(* CODESYS project CtaAppKelvinminuten_1.0.0.0.library
   Description: Kelvinminuten Library der CTA
   Version: 1.0.0.0
   Title: CtaAppKelvinminuten
   Author: SIS
   Company: CTA
   Placeholder: CtaAppKelvinminuten
   DocFormat: reStructuredText
   CompiledLibraryCompatibilityVersion: CODESYS V3.5 SP16 Patch 3
   LanguageModelAttribute: qualified-access-only
   DefaultNamespace: CtaAppKelvinminuten

Project tree, tasks and I/O mapping:
  libraries: CmpBitmapPool, 3.5.17.0 (System); CtaVisSymbols, 1.0.0.0 (CTA); CtaSysConfig, 1.0.0.0 (CTA); CtaAppTime, 1.0.0.0 (CTA); VisuSymbols, 4.5.0.0 (System)
  40 Visualizations/
    visualisation visKelvinminuten
    visualisation popUpKelvinminuten
  30 Program Organization Units/
    function block fbKelvinminuten [ST]: actParameter
  00000000-0000-0000-0000-000000000000|D:\CoDeSys\LibrariesV3\trunk\Intern\CAA\CAA Template\3.4.0.0 draft\Placeholder.xml
  00000000-0000-0000-0000-000000000000|D:\CoDeSys\LibrariesV3\trunk\Intern\CAA\CAA Template\3.2.0.3 draft\Prefix.pdf
  00000000-0000-0000-0000-000000000000|D:\CoDeSys\LibrariesV3\trunk\Intern\CAA\CAA Template\3.5.2.0 draft\Placeholder.xml
  20 Structs/
    data type scParameter
    data type enState
  50 Images/
  10 Documenation/
    global variables VersionHistory
    global variables readMe
  21 Interface/
  11 Library Parameter/
  12 Konstanten/
  60 Textlisten/
  13 Globale Variablen/
  5ce3da45-db07-42e7-a21c-a00fff4ed8f6|Icons\alert.svg
  5ce3da45-db07-42e7-a21c-a00fff4ed8f6|Icons\arrow-down.svg
  5ce3da45-db07-42e7-a21c-a00fff4ed8f6|Icons\arrow-down_square.svg
  5ce3da45-db07-42e7-a21c-a00fff4ed8f6|Icons\arrow-left_solo_black.svg
  5ce3da45-db07-42e7-a21c-a00fff4ed8f6|Icons\arrow-right_solo_black.svg
  5ce3da45-db07-42e7-a21c-a00fff4ed8f6|Icons\arrow-up.svg
  5ce3da45-db07-42e7-a21c-a00fff4ed8f6|Icons\calendar-range.svg
  5ce3da45-db07-42e7-a21c-a00fff4ed8f6|Icons\check.svg
  5ce3da45-db07-42e7-a21c-a00fff4ed8f6|Icons\clock-outline.svg
  5ce3da45-db07-42e7-a21c-a00fff4ed8f6|Icons\close_solo_black.svg
  5ce3da45-db07-42e7-a21c-a00fff4ed8f6|Icons\CtaInfo.svg
  5ce3da45-db07-42e7-a21c-a00fff4ed8f6|Icons\database_black.svg
  5ce3da45-db07-42e7-a21c-a00fff4ed8f6|Icons\delete_solo_black.svg
  5ce3da45-db07-42e7-a21c-a00fff4ed8f6|Icons\engine.svg
  5ce3da45-db07-42e7-a21c-a00fff4ed8f6|Icons\front_hand_Black.svg
  5ce3da45-db07-42e7-a21c-a00fff4ed8f6|Icons\front_hand_Yellow_Off.svg
  5ce3da45-db07-42e7-a21c-a00fff4ed8f6|Icons\gear.svg
  5ce3da45-db07-42e7-a21c-a00fff4ed8f6|Icons\home.svg
  5ce3da45-db07-42e7-a21c-a00fff4ed8f6|Icons\information-variant.svg
  5ce3da45-db07-42e7-a21c-a00fff4ed8f6|Icons\lightning-bolt-circle.svg
  5ce3da45-db07-42e7-a21c-a00fff4ed8f6|Icons\message.svg
  5ce3da45-db07-42e7-a21c-a00fff4ed8f6|Icons\message-alert-variant.svg
  5ce3da45-db07-42e7-a21c-a00fff4ed8f6|Icons\minus_solo_black.svg
  5ce3da45-db07-42e7-a21c-a00fff4ed8f6|Icons\plus_solo_black.svg
  5ce3da45-db07-42e7-a21c-a00fff4ed8f6|Icons\power_solo_black.svg
  5ce3da45-db07-42e7-a21c-a00fff4ed8f6|Icons\refresh_solo_black.svg
  5ce3da45-db07-42e7-a21c-a00fff4ed8f6|Icons\SearchFilter.svg
  5ce3da45-db07-42e7-a21c-a00fff4ed8f6|Icons\signal-celular-alt.svg
  5ce3da45-db07-42e7-a21c-a00fff4ed8f6|Icons\toggle-switch.svg
  5ce3da45-db07-42e7-a21c-a00fff4ed8f6|Icons\Modbus_Organization_Logo.svg
  5ce3da45-db07-42e7-a21c-a00fff4ed8f6|Icons\CheckboxUnchecked_withe.svg
  5ce3da45-db07-42e7-a21c-a00fff4ed8f6|Icons\lock_open_black.svg
  5ce3da45-db07-42e7-a21c-a00fff4ed8f6|Icons\check_green.svg
  5ce3da45-db07-42e7-a21c-a00fff4ed8f6|Icons\filter_black.svg
  5ce3da45-db07-42e7-a21c-a00fff4ed8f6|Icons\CtaLogo.png
  5ce3da45-db07-42e7-a21c-a00fff4ed8f6|Icons\Grafana_Logo.svg
  5ce3da45-db07-42e7-a21c-a00fff4ed8f6|Icons\hourglass_top.svg
  text list GlobalTextList
*)

// 20 Structs/scParameter
TYPE scParameter :
	STRUCT
		fbrKmZuschalt   : CtaSysConfig.fbREAL;
		fbrKmWegschalt  : CtaSysConfig.fbREAL;
		fbrDiffFastExit : CtaSysConfig.fbREAL;
		fbrHysterese    : CtaSysConfig.fbREAL;
		fbiMaxStufen    : CtaSysConfig.fbINT;
		fbiMinStufen    : CtaSysConfig.fbINT;
	END_STRUCT
END_TYPE

// 20 Structs/enState
TYPE enState :
(
	AUS                   	:= 0,
    KEIN_BEDARF           	:= 1,
    LOCKDOWN              	:= 2,
    GAS_FLUID             	:= 3,
    GAS_AIR               	:= 4,
    UMSCHALTUNG_STOP      	:= 5,
	UMSCHALTUNG_NORMAL		:= 6,
    NICHT_BEREIT          	:= 9,
    KÜHLBETRIEB           	:= 10,
    HEIZBETRIEB           	:= 20,
	HEIZBETRIEB2			:= 21,
    BWWBETRIEB            	:= 30,
    REVERSIBEL            	:= 40,
    FREECOOL              	:= 50
);
END_TYPE

// 10 Documenation/VersionHistory
(* 

.. image:: ../../Images/CTA_Logo.jpg
   :align: right
   :width: 15% 

**Vorlage**   


============ =========== =========== ============================================
**Date**     **Version** **Author**  **Change**
------------ ----------- ----------- --------------------------------------------
04.03.2021   0.0.0.0     SIS         Vorlage erstellt

============ =========== =========== ============================================


*)
VAR_GLOBAL
    stInfo : STRING:= '0.0.0.0, Vorlage, CTA';
END_VAR

// 10 Documenation/readMe
(*

**ReadMe**
 
|	**Empfehlung**
|
|	Die Bibliothek CtaAppKelvinminuten dient der Berechnung der geforderten Stufen unter Berücksichtigung des Soll und Istwertes und der Konfigurierten Stufen.
|	Instanzieren Sie den CtaAppKelvinminuten.fbKelvinminuten in ihrem Funktionsbaustein oder POU beispielsweise als fbStufen oder beliebig.
|	Deklarieren Sie die Struktur Variable welche als Parameter und zur ansteuerung dienen wie im Code beispiel.
|  
| *Beispiel* 

+-----------------------+---------------------------------------------------------------------------------------------------------------------------------------------------------------------------------------------------------------------------------------------------------------------------------------------------------------------------------------------------------------------------------------------------------------------------------------+
| Beschreibung          |  Code                                                                                                                                                                                                                                                                                                                                                                                                                                 |
+=======================+=======================================================================================================================================================================================================================================================================================================================================================================================================================================+
| Pou oder SmFb         | .. code-block:: codesys                                                                                                                                                                                                                                                                                                                                                                                                               |
|                       |                                                                                                                                                                                                                                                                                                                                                                                                                                       |
|                       |	// Deklaration als VAR im POU oder dem selbsterstellten Funktionsbaustein                                                                                                                                                                                                                                                                                                                                                       	|
|                       |   VAR   																																																																																																								|
|						|	    (*Stufenschaltung*)																																																		 																																																		|
|						|		fbStufen			: CtaAppKelvinminuten.fbKelvinminuten;                                                                                                                                                                                                                                                                                                                                                              		|
|						|																																																																																																										|
+-----------------------+---------------------------------------------------------------------------------------------------------------------------------------------------------------------------------------------------------------------------------------------------------------------------------------------------------------------------------------------------------------------------------------------------------------------------------------+
| Code für Init         | .. code-block:: codesys                                                                                                                                                                                                                                                                                                                                                                                                               |
|                       |   																																																																																																									|
| 						|	// Kopieren des nachfolgenden Codes in eine Action zur Initialisierung der Parameter. Zum Beispiel actConfig.																																																																														|
|                       |	{region " Stufenschaltung "}                                                                                                                                                                                                                                                                                                                                                                                                     	|
| 						|		(*Basis*)																																																																																																						|
|						|		fbStufen.scParameter.fbrKmZuschalt               		(_wertInit :=	  5000		, _minInit :=			, _maxInit :=			);		//P1 Wert nach welchem eine Stufe zugeschalten wird																																																									|
|						|		fbStufen.scParameter.fbrKmWegschalt						(_wertInit :=	  2000		, _minInit :=			, _maxInit :=			);		//P2 Wert nach welchem eine Stufe weggeschalten wird																																																								| 
|						|		fbStufen.scParameter.fbrDiffFastExit					(_wertInit :=	  1000		, _minInit :=			, _maxInit :=			);		//P3 Differenz welche eine sofortige Wegschaltung bewirkt.																																																							| 
|						|		fbStufen.scParameter.fbrHysterese						(_wertInit :=		50		, _minInit :=			, _maxInit := 			);		//P4 Einstellbare Hysterese für zu und Wegschaltung																																																									| 
|						|		fbStufen.scParameter.fbiMinStufen						(_wertInit := 		 1		, _minInit :=   		, _maxInit := 			);		//P5 Minimal mögliche Anzahl Stufen																																																													|
|						|		fbStufen.scParameter.fbiMaxStufen						(_wertInit := 		 4		, _minInit :=			, _maxInit := 			);		//P6 Maximal mögliche Anzahl 																																																														|
|						|	{endregion}                                                                                                                                                      																																																																	| 
+-----------------------+---------------------------------------------------------------------------------------------------------------------------------------------------------------------------------------------------------------------------------------------------------------------------------------------------------------------------------------------------------------------------------------------------------------------------------------+
*)                                                                                                                                                                                                                                                                                                                                                                                                                                                               
 VAR_GLOBAL                                                                                                                                                                                                                                                                                                                                                                                                                                                      
    xReadMeDone              :   BOOL;                                                                                                                                                                                                                                                                                                                                                                                                                           
END_VAR

// 30 Program Organization Units/fbKelvinminuten
FUNCTION_BLOCK fbKelvinminuten
VAR_INPUT
	xEn             : BOOL;                     // Freigabe Kmin rechnung
    xReadyRelease   : BOOL;                     // Freigabe Zuschaltung
	xInvert			: BOOL;						// Invertierung der Wertberechnung
    rIst            : REAL;                     // Istwert
    rSoll           : REAL;                     // Sollwert
END_VAR
VAR_OUTPUT
	iStufen         : INT;                      // Angeforderte Stufen
END_VAR
VAR
	rKmZuschalt     : REAL;
    rKmWegschalt    : REAL;
    rCycleTime      : REAL;
	fbCycle			: CtaAppTime.fbTimeMeasurement;	
    fbConfigFile    : CtaSysConfig.fbConfigFile;
	scParameter		: scParameter;
END_VAR

actParameter();
// Zykluszeit erkennen
rCycleTime  :=  LTIME_TO_REAL(fbCycle.stop())/1000000000; // Ltime to ms
fbCycle.Start();
// Freigabe 
IF xEn AND rCycleTime <> 0 THEN
	
	IF NOT xInvert THEN
	
		// Zuschalten
		IF rIst > rSoll + scParameter.fbrHysterese.proValue AND (iStufen < scParameter.fbiMaxStufen.proValue OR scParameter.fbiMaxStufen.proValue = 0 ) THEN
			rKmWegschalt := 0; // Wegschaltung reset
			rKmZuschalt  := rKmZuschalt + ((rIst-rSoll)*rCycleTime/60);
		// Wegschalten
		ELSIF rIst < rSoll - scParameter.fbrHysterese.proValue AND (iStufen > scParameter.fbiMinStufen.proValue OR scParameter.fbiMinStufen.proValue = 0 ) THEN
			rKmZuschalt := 0; // Zuschaltung reset
			rKmWegschalt:= rKmWegschalt + ((rSoll-rIst)*rCycleTime/60);
		END_IF; 
		// Stufen wegschalten wenn abweichung grösser als fast Exit
		IF rIst < rSoll - scParameter.fbrDiffFastExit.proValue THEN
			rKmZuschalt     := 0;
			rKmWegschalt    := 0;
			iStufen         := iStufen -1;   
		// Stufen Zuschalten wenn Km > zuschalt Km & Bereit zum zuschalten    
		ELSIF rKmZuschalt >= scParameter.fbrKmZuschalt.proValue AND xReadyRelease THEN
			rKmZuschalt     := 0;
			iStufen         := iStufen + 1;
		// Stufen Wegschalten wenn Km > wegschalt Km & Bereit zum zuschalten    
		ELSIF rKmWegschalt >= scParameter.fbrKmWegschalt.proValue THEN    
			rKmWegschalt    := 0;
			iStufen         := iStufen - 1;
		END_IF;
		// Limitierung Min & Max Stufen
		IF scParameter.fbiMinStufen.proValue <> scParameter.fbiMaxStufen.proValue THEN
			iStufen := LIMIT(scParameter.fbiMinStufen.proValue,iStufen,scParameter.fbiMaxStufen.proValue);    
		ELSE
			iStufen := MAX(0,iStufen);
		END_IF;		
	ELSE		
		// Zuschalten
		IF rIst < rSoll - scParameter.fbrHysterese.proValue AND (iStufen < scParameter.fbiMaxStufen.proValue OR scParameter.fbiMaxStufen.proValue = 0 ) THEN
			rKmWegschalt := 0; // Wegschaltung reset
			rKmZuschalt  := rKmZuschalt + ((rSoll-rIst)*rCycleTime/60);
		// Wegschalten
		ELSIF rIst > rSoll + scParameter.fbrHysterese.proValue AND (iStufen > scParameter.fbiMinStufen.proValue OR scParameter.fbiMinStufen.proValue = 0 ) THEN
			rKmZuschalt := 0; // Zuschaltung reset
			rKmWegschalt:= rKmWegschalt + ((rIst-rSoll)*rCycleTime/60);
		END_IF; 
		// Stufen wegschalten wenn abweichung grösser als fast Exit
		IF rIst > rSoll + scParameter.fbrDiffFastExit.proValue THEN
			rKmZuschalt     := 0;
			rKmWegschalt    := 0;
			iStufen         := iStufen -1;   
		// Stufen Zuschalten wenn Km > zuschalt Km & Bereit zum zuschalten    
		ELSIF rKmZuschalt >= scParameter.fbrKmZuschalt.proValue AND xReadyRelease THEN
			rKmZuschalt     := 0;
			iStufen         := iStufen + 1;
		// Stufen Wegschalten wenn Km > wegschalt Km & Bereit zum zuschalten    
		ELSIF rKmWegschalt >= scParameter.fbrKmWegschalt.proValue THEN    
			rKmWegschalt    := 0;
			iStufen         := iStufen - 1;
		END_IF;
		// Limitierung Min & Max Stufen
		IF scParameter.fbiMinStufen.proValue <> scParameter.fbiMaxStufen.proValue THEN
			iStufen := LIMIT(scParameter.fbiMinStufen.proValue,iStufen,scParameter.fbiMaxStufen.proValue);    
		ELSE
			iStufen := MAX(0,iStufen);
		END_IF;
	END_IF
	
// Reset wenn ausgeschalten    
ELSE
    iStufen         := 0; 
    rKmWegschalt    := 0;  
    rKmZuschalt     := 0; 
END_IF;

ACTION actParameter:
fbConfigFile();

scParameter.fbrKmZuschalt   (_usiParaNr := 1, itfConfigFb := fbConfigFile); // Zuschalt Kelvin Minuten
scParameter.fbrKmWegschalt  (_usiParaNr := 2, itfConfigFb := fbConfigFile); // Wegschalt Kelvin Minute
scParameter.fbrDiffFastExit (_usiParaNr := 3, itfConfigFb := fbConfigFile); // Differenz Lastabwurf
scParameter.fbrHysterese    (_usiParaNr := 4, itfConfigFb := fbConfigFile); // Hysterese für Zu & Wegschalt rechnung
scParameter.fbiMinStufen	(_usiParaNr := 5, itfConfigFb := fbConfigFile); // Minimum Stufen
scParameter.fbiMaxStufen	(_usiParaNr := 6, itfConfigFb := fbConfigFile); // Maximum Stufen
END_ACTION

END_FUNCTION_BLOCK

// 40 Visualizations/visKelvinminuten
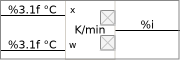
VISUALIZATION visKelvinminuten  // 180x60
VAR_IN_OUT
	fbKelvinminutenIN	: fbKelvinminuten;
END_VAR
    Textfield (115,20 65x10), "%i", text variable: fbKelvinminutenIN.iStufen
    Textfield (0,5 65x10), "%3.1f °C", text variable: fbKelvinminutenIN.rIst
    Textfield (0,40 65x10), "%3.1f °C", text variable: fbKelvinminutenIN.rSoll
    Line (115,30) (180,30)
    Line (0,50) (65,50)
    Line (0,15) (65,15)
    Textfield (65,0 50x60), "K/min"
        OnMouseClick:  Dialog=popUpKelvinminuten, Parameters={fbKelvinminutenIN: fbKelvinminutenIN}, Selected={1: }, OpenModal=True, OpenCentered=True
    Label (68,5 10x10), "x"
    Label (68,40 10x10), "w"
    Image (100,10 15x15), invisible if: fbKelvinminutenIN.scParameter.fbrKmZuschalt.rValue = 0, image: LibVis01VisuBasic.imgpVisuCTA.plus_solo_black
    Image (100,35 15x15), invisible if: fbKelvinminutenIN.scParameter.fbrKmWegschalt.rValue = 0, image: LibVis01VisuBasic.imgpVisuCTA.minus_solo_black
END_VISUALIZATION

// 40 Visualizations/popUpKelvinminuten
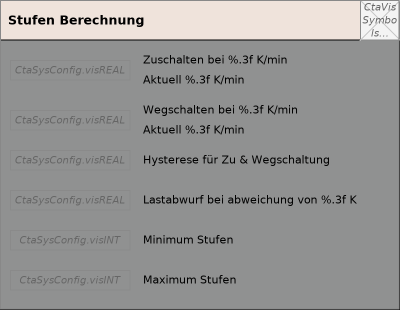
VISUALIZATION popUpKelvinminuten  // 400x310
VAR_IN_OUT
	{attribute 'VAR_IN_OUT_AS_POINTER'}
	fbKelvinminutenIN	:	fbKelvinminuten;
END_VAR
    Rectangle (0,0 400x310)
    Rectangle (0,0 400x40)
    Label (5,10 150x20), "Stufen Berechnung"
    Frame (10,60 120x20)
        shows CtaSysConfig.visREAL(visfbREALIn := fbKelvinminutenIN.scParameter.fbrKmZuschalt, stPhysikalischeEinheit := 'K/min')
    Textfield (140,70 200x20), "Aktuell %.3f K/min", text variable: fbKelvinminutenIN.rKmZuschalt
    Frame (10,110 120x20)
        shows CtaSysConfig.visREAL(visfbREALIn := fbKelvinminutenIN.scParameter.fbrKmWegschalt, stPhysikalischeEinheit := 'K/min')
    Textfield (140,120 200x20), "Aktuell %.3f K/min", text variable: fbKelvinminutenIN.rKmWegschalt
    Frame (10,150 120x20)
        shows CtaSysConfig.visREAL(visfbREALIn := fbKelvinminutenIN.scParameter.fbrHysterese, stPhysikalischeEinheit := 'K')
    Label (140,150 220x20), "Hysterese für Zu & Wegschaltung"
    Frame (10,190 120x20)
        shows CtaSysConfig.visREAL(visfbREALIn := fbKelvinminutenIN.scParameter.fbrDiffFastExit, stPhysikalischeEinheit := 'K')
    Frame (10,230 120x20)
        shows CtaSysConfig.visINT(visfbINTIn := fbKelvinminutenIN.scParameter.fbiMinStufen)
    Label (140,230 150x20), "Minimum Stufen"
    Frame (10,270 120x20)
        shows CtaSysConfig.visINT(visfbINTIn := fbKelvinminutenIN.scParameter.fbiMaxStufen)
    Label (140,270 150x20), "Maximum Stufen"
    Image (360,0 40x40), image: CtaVisSymbols.ImagePool.close_solo_black
        OnMouseUp:  Dialog=popUpKelvinMinuten, Result=None, NumpadKeypadSet=True
    Textfield (140,50 200x20), "Zuschalten bei %.3f K/min", text variable: fbKelvinminutenIN.scParameter.fbrKmZuschalt.rValue
    Textfield (140,100 200x20), "Wegschalten bei %.3f K/min", text variable: fbKelvinminutenIN.scParameter.fbrKmWegschalt.rValue
    Textfield (140,190 258x20), "Lastabwurf bei abweichung von %.3f K", text variable: fbKelvinminutenIN.scParameter.fbrDiffFastExit.rValue
END_VISUALIZATION
